// Mitsubishi GX Works2 project: BookEX6_31 Rotation   PLC: Q13UDV

TYPE WordBit : STRUCT
  Data : DWORD;
  Flag : BOOL;
END_STRUCT END_TYPE

// global labels: Global
VAR_GLOBAL
  bVar0 AT M5000 : BOOL;
  abArray0 AT M5010 : ARRAY [0..49] OF BOOL;
  sStr0 AT D5000 : STRING[199];
  sStr1 AT D5100 : STRING[199];
  sStr2 AT D5200 : STRING[199];
  sStr3 AT D5300 : STRING[199];
  sStr4 AT D5400 : STRING[199];
  sStr5 AT D5500 : STRING[199];
  sStr6 AT D5600 : STRING[199];
  sStr7 AT D5700 : STRING[199];
  sStr8 AT D5800 : STRING[199];
  sStr9 AT D5900 : STRING[199];
  iVar0 AT D4500 : INT;
  iVar1 AT D4501 : INT;
  iVar2 AT D4502 : INT;
  iVar3 AT D4503 : INT;
  iVar4 AT D4504 : INT;
  iVar5 AT D4505 : INT;
  iVar6 AT D4506 : INT;
  iVar7 AT D4507 : INT;
  iVar8 AT D4508 : INT;
  iVar9 AT D4509 : INT;
  dVar0 AT D4510 : DINT;
  dVar1 AT D4512 : DINT;
  dVar2 AT D4514 : DINT;
  dVar3 AT D4516 : DINT;
  dVar4 AT D4518 : DINT;
  dVar5 AT D4520 : DINT;
  dVar6 AT D4522 : DINT;
  dVar7 AT D4524 : DINT;
  dVar8 AT D4526 : DINT;
  dVar9 AT D4528 : DINT;
  wVar0 AT D4530 : WORD;
  wVar1 AT D4531 : WORD;
  wVar2 AT D4532 : WORD;
  wVar3 AT D4533 : WORD;
  wVar4 AT D4534 : WORD;
  wVar5 AT D4535 : WORD;
  wVar6 AT D4536 : WORD;
  wVar7 AT D4537 : WORD;
  wVar8 AT D4538 : WORD;
  wVar9 AT D4539 : WORD;
  dwVar0 AT D4540 : DWORD;
  dwVar1 AT D4542 : DWORD;
  dwVar2 AT D4544 : DWORD;
  dwVar3 AT D4546 : DWORD;
  dwVar4 AT D4548 : DWORD;
  dwVar5 AT D4550 : DWORD;
  dwVar6 AT D4552 : DWORD;
  dwVar7 AT D4554 : DWORD;
  dwVar8 AT D4556 : DWORD;
  dwVar9 AT D4558 : DWORD;
  fsVar0 AT D4560 : REAL;
  fsVar1 AT D4562 : REAL;
  fsVar2 AT D4564 : REAL;
  fsVar3 AT D4566 : REAL;
  fsVar4 AT D4568 : REAL;
  fsVar5 AT D4570 : REAL;
  fsVar6 AT D4572 : REAL;
  fsVar7 AT D4574 : REAL;
  fsVar8 AT D4576 : REAL;
  fsVar9 AT D4578 : REAL;
  fdVar0 AT D4580 : LREAL;
  tTime0 AT D4620 : TIME;
  tTime1 AT D4622 : TIME;
  tTime2 AT D4624 : TIME;
  tTime3 AT D4626 : TIME;
  tTime4 AT D4628 : TIME;
  tTime5 AT D4630 : TIME;
  tTime6 AT D4632 : TIME;
  tTime7 AT D4634 : TIME;
  tTime8 AT D4636 : TIME;
  tTime9 AT D4638 : TIME;
  tTime10 AT D4640 : TIME;
  bVar1 AT M5001 : BOOL;
  bVar2 AT M5002 : BOOL;
  bVar3 AT M5003 : BOOL;
  bVar4 AT M5004 : BOOL;
  bVar5 AT M5005 : BOOL;
  bVar6 AT M5006 : BOOL;
  bVar7 AT M5007 : BOOL;
  bVar8 AT M5008 : BOOL;
  bVar9 AT M5009 : BOOL;
  abArray1 AT M5060 : ARRAY [0..49] OF BOOL;
  abArray2 AT M5110 : ARRAY [0..49] OF BOOL;
  abArray3 AT M5160 : ARRAY [0..49] OF BOOL;
  abArray4 AT M5210 : ARRAY [0..49] OF BOOL;
  abArray5 AT M5260 : ARRAY [0..49] OF BOOL;
  abArray6 AT M5310 : ARRAY [0..49] OF BOOL;
  abArray7 AT M5360 : ARRAY [0..49] OF BOOL;
  abArray8 AT M5410 : ARRAY [0..49] OF BOOL;
  abArray9 AT M5460 : ARRAY [0..49] OF BOOL;
  fdVar1 AT D4584 : LREAL;
  fdVar2 AT D4588 : LREAL;
  fdVar3 AT D4592 : LREAL;
  fdVar4 AT D4596 : LREAL;
  fdVar5 AT D4600 : LREAL;
  fdVar6 AT D4604 : LREAL;
  fdVar7 AT D4608 : LREAL;
  fdVar8 AT D4612 : LREAL;
  fdVar9 AT D4616 : LREAL;
  afsPen0 AT D2000 : ARRAY [0..499] OF REAL;
  afsPen1 AT D3000 : ARRAY [0..499] OF REAL;
END_VAR
// user libraries (not included): HMI

FUNCTION BitLoadPos2
VAR_INPUT
  w_IN : WORD;
END_VAR
VAR
  wTmp1 : WORD;
END_VAR
VAR_INPUT
  b_Val : BOOL;
  i_Pos : INT;
  i_No : INT;
END_VAR
VAR
  wTmp2 : WORD;
  wTmp3 : WORD;
END_VAR
;
wTmp1 := HFFFF;
wTmp2 := w_IN;
IF b_Val THEN
	SFR(TRUE, 16 - i_No, wTmp1 );
	ROR(TRUE,  i_Pos, wTmp2);
	wTmp3 := wTmp1 OR wTmp2;
	ROL(TRUE,  i_Pos, wTmp3);
ELSE
	SFL(TRUE,  i_No, wTmp1 );
	ROR(TRUE,  i_Pos, wTmp2);
	wTmp3 := wTmp1 AND wTmp2;
	ROL(TRUE,  i_Pos, wTmp3);
END_IF;
BitLoadPos2 := wTmp3;
END_FUNCTION

FUNCTION dwBitArray
VAR_INPUT
  dwInp : DWORD;
  iOffset : INT;
  iLength : INT;
END_VAR
VAR
  ix : INT;
  dwData : DWORD;
  dwMask : DWORD;
END_VAR
;
dwMask := 0;
FOR ix := 0 TO iLength-1 DO 
	SM700 := TRUE;
	DRCL(TRUE, 1, dwMask); 
END_FOR;
dwData := dwInp;
DROR(TRUE, iOffset, dwData);
dwBitArray := dwData AND dwMask;
END_FUNCTION

PROGRAM ExBitArray
(* structured ladder/FBD written out as ST: instructions are called as NAME(EN, inputs, outputs); _pN, _eN, _tN stand for wires *)
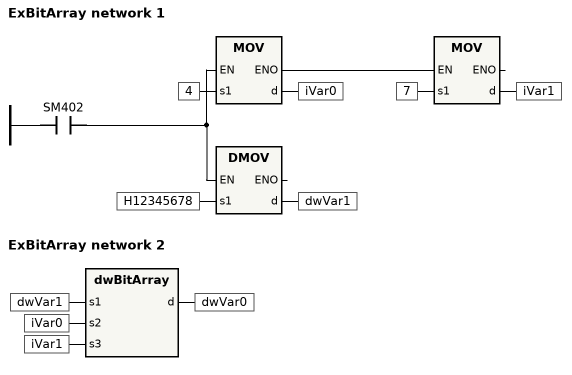
(* network 1 *)
_e1 := MOV(SM402, 4, iVar0);
MOV(_e1, 7, iVar1);
DMOV(SM402, H12345678, dwVar1);
(* network 2 *)
dwVar0 := dwBitArray(dwVar1, iVar0, iVar1);
END_PROGRAM

PROGRAM ExStandard
VAR
  Mov8WORD_1 : Mov8WORD;
  Mov8DWORD_1 : Mov8DWORD;
  wTst0 : WORD;
  wTst1 : WORD;
  wTst2 : WORD;
  wTst3 : WORD;
  wTst4 : WORD;
  dwTst0 : DWORD;
  dwTst1 : DWORD;
  dwTst2 : DWORD;
  dwTst3 : DWORD;
  dwTst4 : DWORD;
  wTst5 : WORD;
  wTst6 : WORD;
  wTst7 : WORD;
  dwTst5 : DWORD;
  dwTst6 : DWORD;
  dwTst7 : DWORD;
END_VAR
(* structured ladder/FBD written out as ST: instructions are called as NAME(EN, inputs, outputs); _pN, _eN, _tN stand for wires *)
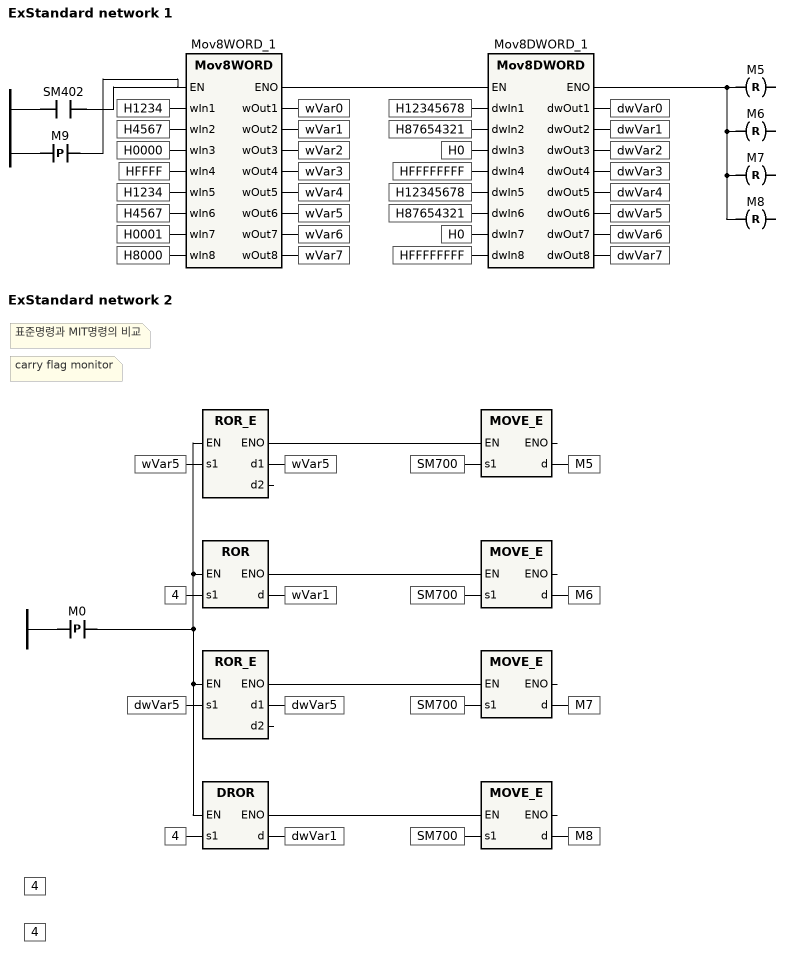
(* network 1 *)
Mov8WORD_1(EN := SM402 OR LDP(TRUE, M9), wIn1 := H1234, wIn2 := H4567, wIn3 := H0000, wIn4 := HFFFF, wIn5 := H1234, wIn6 := H4567, wIn7 := H0001, wIn8 := H8000, wOut1 => wVar0, wOut2 => wVar1, wOut3 => wVar2, wOut4 => wVar3, wOut5 => wVar4, wOut6 => wVar5, wOut7 => wVar6, wOut8 => wVar7);
Mov8DWORD_1(EN := Mov8WORD_1.ENO, dwIn1 := H12345678, dwIn2 := H87654321, dwIn3 := H0, dwIn4 := HFFFFFFFF, dwIn5 := H12345678, dwIn6 := H87654321, dwIn7 := H0, dwIn8 := HFFFFFFFF, dwOut1 => dwVar0, dwOut2 => dwVar1, dwOut3 => dwVar2, dwOut4 => dwVar3, dwOut5 => dwVar4, dwOut6 => dwVar5, dwOut7 => dwVar6, dwOut8 => dwVar7);
RST(Mov8DWORD_1.ENO, M5);
RST(Mov8DWORD_1.ENO, M6);
RST(Mov8DWORD_1.ENO, M7);
RST(Mov8DWORD_1.ENO, M8);
(* network 2 *)
(* 표준명령과 MIT명령의 비교 *)
(* carry flag monitor *)
_p1 := LDP(TRUE, M0);
_e2 := ROR_E(_p1, wVar5, wVar5, _open);
MOVE_E(_e2, SM700, M5);
_e3 := ROR(_p1, 4, wVar1);
MOVE_E(_e3, SM700, M6);
_e4 := ROR_E(_p1, dwVar5, dwVar5, _open);
MOVE_E(_e4, SM700, M7);
_e5 := DROR(_p1, 4, dwVar1);
MOVE_E(_e5, SM700, M8);
(* not connected to any output: 4, 4 *)
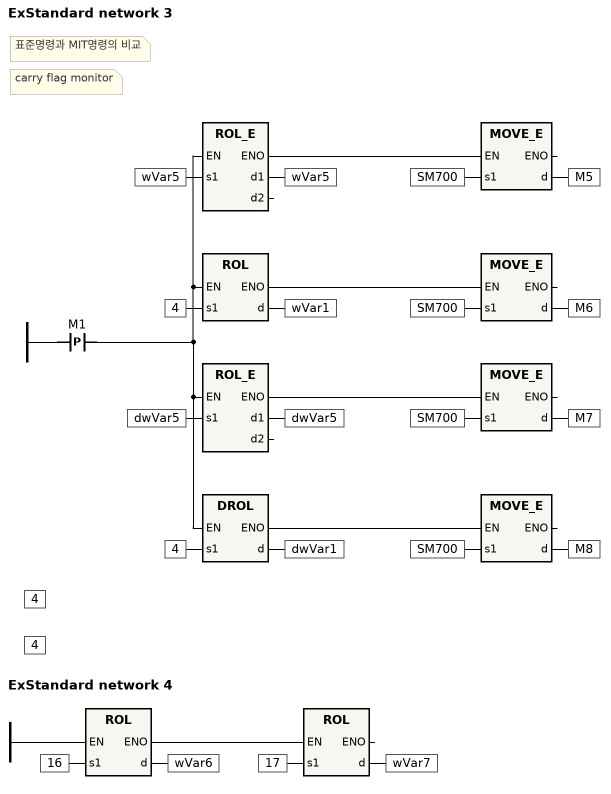
(* network 3 *)
(* 표준명령과 MIT명령의 비교 *)
(* carry flag monitor *)
_p1 := LDP(TRUE, M1);
_e2 := ROL_E(_p1, wVar5, wVar5, _open);
MOVE_E(_e2, SM700, M5);
_e3 := ROL(_p1, 4, wVar1);
MOVE_E(_e3, SM700, M6);
_e4 := ROL_E(_p1, dwVar5, dwVar5, _open);
MOVE_E(_e4, SM700, M7);
_e5 := DROL(_p1, 4, dwVar1);
MOVE_E(_e5, SM700, M8);
(* not connected to any output: 4, 4 *)
(* network 4 *)
_e1 := ROL(TRUE, 16, wVar6);
ROL(_e1, 17, wVar7);
END_PROGRAM

PROGRAM ExDROR
VAR
  Mov8WORD_1 : Mov8WORD;
  Mov8DWORD_1 : Mov8DWORD;
  wTst0 : WORD;
  wTst1 : WORD;
  wTst2 : WORD;
  wTst3 : WORD;
  wTst4 : WORD;
  dwTst0 : DWORD;
  dwTst1 : DWORD;
  dwTst2 : DWORD;
  dwTst3 : DWORD;
  dwTst4 : DWORD;
END_VAR
(* structured ladder/FBD written out as ST: instructions are called as NAME(EN, inputs, outputs); _pN, _eN, _tN stand for wires *)
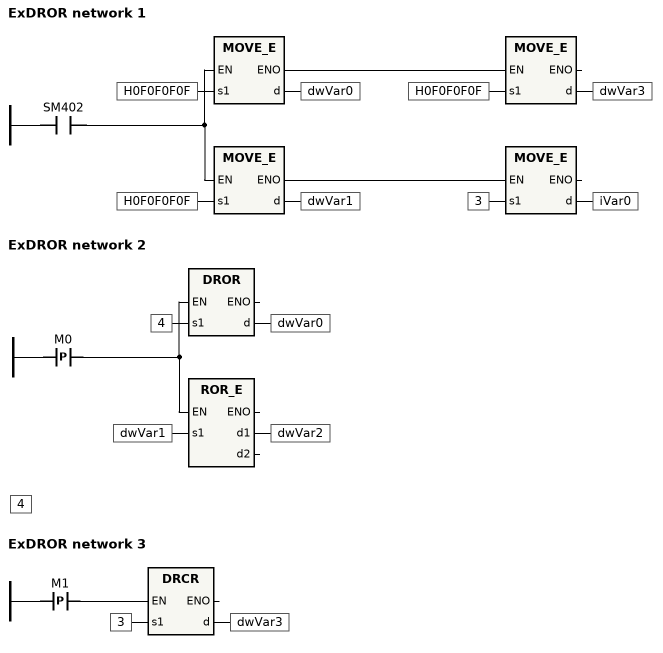
(* network 1 *)
_e1 := MOVE_E(SM402, H0F0F0F0F, dwVar0);
MOVE_E(_e1, H0F0F0F0F, dwVar3);
_e2 := MOVE_E(SM402, H0F0F0F0F, dwVar1);
MOVE_E(_e2, 3, iVar0);
(* network 2 *)
_p1 := LDP(TRUE, M0);
DROR(_p1, 4, dwVar0);
ROR_E(_p1, dwVar1, dwVar2, _open);
(* not connected to any output: 4 *)
(* network 3 *)
DRCR(LDP(TRUE, M1), 3, dwVar3);
END_PROGRAM

PROGRAM ExLib
(* structured ladder/FBD written out as ST: instructions are called as NAME(EN, inputs, outputs); _pN, _eN, _tN stand for wires *)
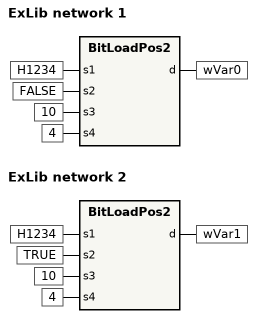
(* network 1 *)
wVar0 := BitLoadPos2(H1234, FALSE, 10, 4);
(* network 2 *)
wVar1 := BitLoadPos2(H1234, TRUE, 10, 4);
END_PROGRAM

PROGRAM ExRingCnt
VAR
  TON_E_1 : TON_E;
  HMI05_1 : HMI05;
END_VAR
(* structured ladder/FBD written out as ST: instructions are called as NAME(EN, inputs, outputs); _pN, _eN, _tN stand for wires *)
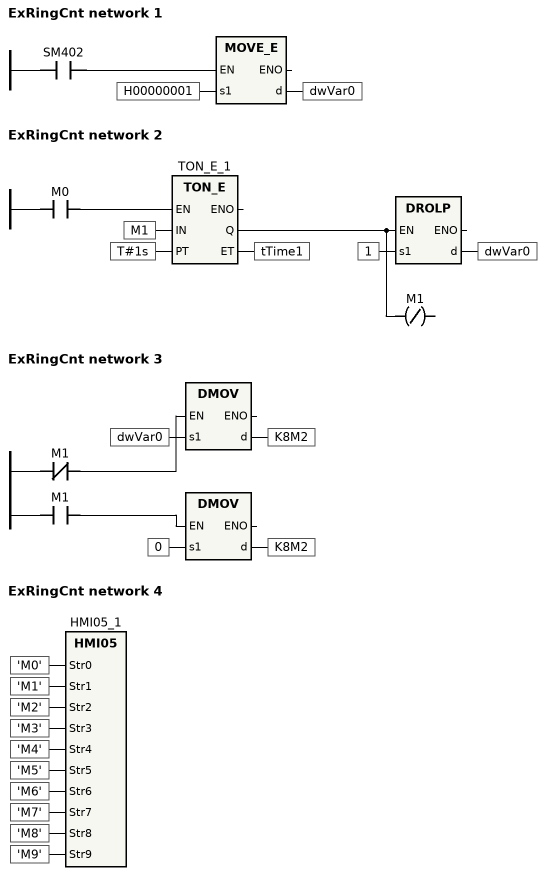
(* network 1 *)
MOVE_E(SM402, H00000001, dwVar0);
(* network 2 *)
TON_E_1(EN := M0, IN := M1, PT := T#1s, ET => tTime1);
M1 := NOT TON_E_1.Q;
DROLP(TON_E_1.Q, 1, dwVar0);
(* network 3 *)
DMOV(NOT M1, dwVar0, K8M2);
DMOV(M1, 0, K8M2);
(* network 4 *)
HMI05_1(Str0 := 'M0', Str1 := 'M1', Str2 := 'M2', Str3 := 'M3', Str4 := 'M4', Str5 := 'M5', Str6 := 'M6', Str7 := 'M7', Str8 := 'M8', Str9 := 'M9');
END_PROGRAM

PROGRAM ExROL
VAR
  Mov8WORD_1 : Mov8WORD;
  Mov8DWORD_1 : Mov8DWORD;
  wTst0 : WORD;
  wTst1 : WORD;
  wTst2 : WORD;
  wTst3 : WORD;
  wTst4 : WORD;
  dwTst0 : DWORD;
  dwTst1 : DWORD;
  dwTst2 : DWORD;
  dwTst3 : DWORD;
  dwTst4 : DWORD;
END_VAR
(* structured ladder/FBD written out as ST: instructions are called as NAME(EN, inputs, outputs); _pN, _eN, _tN stand for wires *)
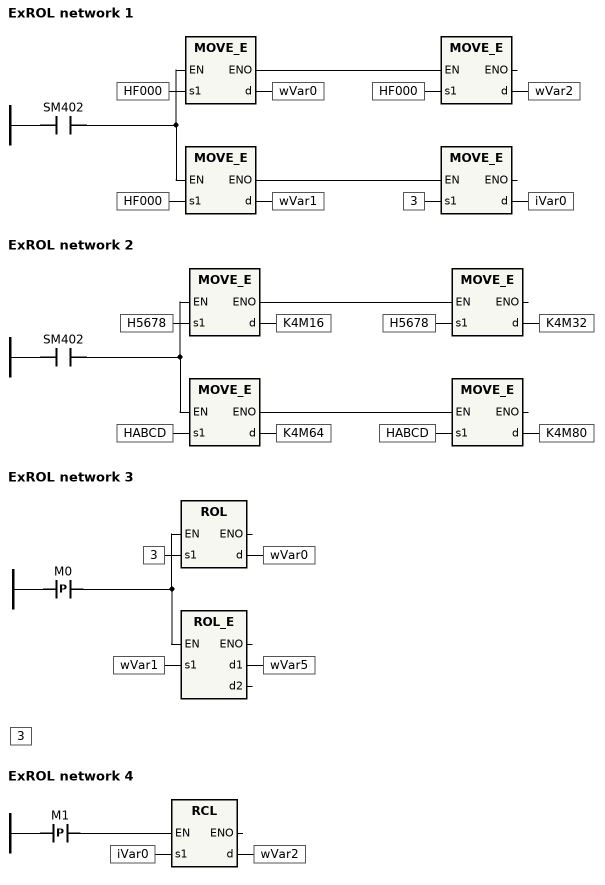
(* network 1 *)
_e1 := MOVE_E(SM402, HF000, wVar0);
MOVE_E(_e1, HF000, wVar2);
_e2 := MOVE_E(SM402, HF000, wVar1);
MOVE_E(_e2, 3, iVar0);
(* network 2 *)
_e1 := MOVE_E(SM402, H5678, K4M16);
MOVE_E(_e1, H5678, K4M32);
_e2 := MOVE_E(SM402, HABCD, K4M64);
MOVE_E(_e2, HABCD, K4M80);
(* network 3 *)
_p1 := LDP(TRUE, M0);
ROL(_p1, 3, wVar0);
ROL_E(_p1, wVar1, wVar5, _open);
(* not connected to any output: 3 *)
(* network 4 *)
RCL(LDP(TRUE, M1), iVar0, wVar2);
END_PROGRAM

PROGRAM ExROR
VAR
  Mov8WORD_1 : Mov8WORD;
  Mov8DWORD_1 : Mov8DWORD;
  wTst0 : WORD;
  wTst1 : WORD;
  wTst2 : WORD;
  wTst3 : WORD;
  wTst4 : WORD;
  dwTst0 : DWORD;
  dwTst1 : DWORD;
  dwTst2 : DWORD;
  dwTst3 : DWORD;
  dwTst4 : DWORD;
END_VAR
(* structured ladder/FBD written out as ST: instructions are called as NAME(EN, inputs, outputs); _pN, _eN, _tN stand for wires *)
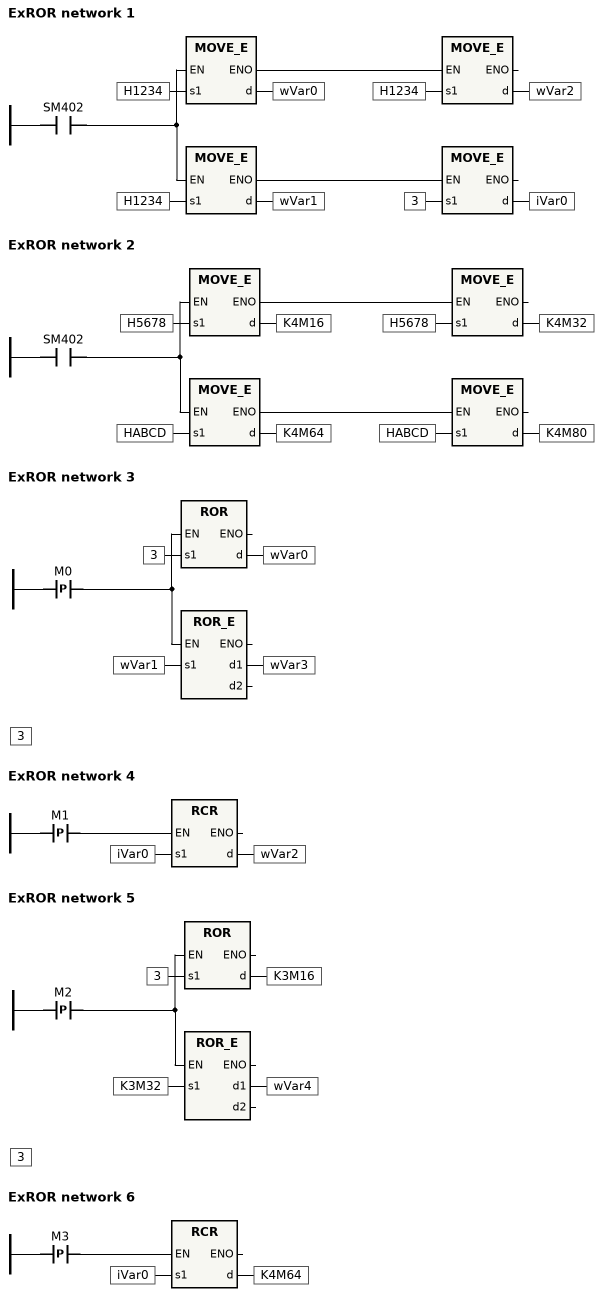
(* network 1 *)
_e1 := MOVE_E(SM402, H1234, wVar0);
MOVE_E(_e1, H1234, wVar2);
_e2 := MOVE_E(SM402, H1234, wVar1);
MOVE_E(_e2, 3, iVar0);
(* network 2 *)
_e1 := MOVE_E(SM402, H5678, K4M16);
MOVE_E(_e1, H5678, K4M32);
_e2 := MOVE_E(SM402, HABCD, K4M64);
MOVE_E(_e2, HABCD, K4M80);
(* network 3 *)
_p1 := LDP(TRUE, M0);
ROR(_p1, 3, wVar0);
ROR_E(_p1, wVar1, wVar3, _open);
(* not connected to any output: 3 *)
(* network 4 *)
RCR(LDP(TRUE, M1), iVar0, wVar2);
(* network 5 *)
_p1 := LDP(TRUE, M2);
ROR(_p1, 3, K3M16);
ROR_E(_p1, K3M32, wVar4, _open);
(* not connected to any output: 3 *)
(* network 6 *)
RCR(LDP(TRUE, M3), iVar0, K4M64);
END_PROGRAM

PROGRAM ExDROL
VAR
  Mov8WORD_1 : Mov8WORD;
  Mov8DWORD_1 : Mov8DWORD;
  wTst0 : WORD;
  wTst1 : WORD;
  wTst2 : WORD;
  wTst3 : WORD;
  wTst4 : WORD;
  dwTst0 : DWORD;
  dwTst1 : DWORD;
  dwTst2 : DWORD;
  dwTst3 : DWORD;
  dwTst4 : DWORD;
  TON_E_1 : TON_E;
END_VAR
(* structured ladder/FBD written out as ST: instructions are called as NAME(EN, inputs, outputs); _pN, _eN, _tN stand for wires *)
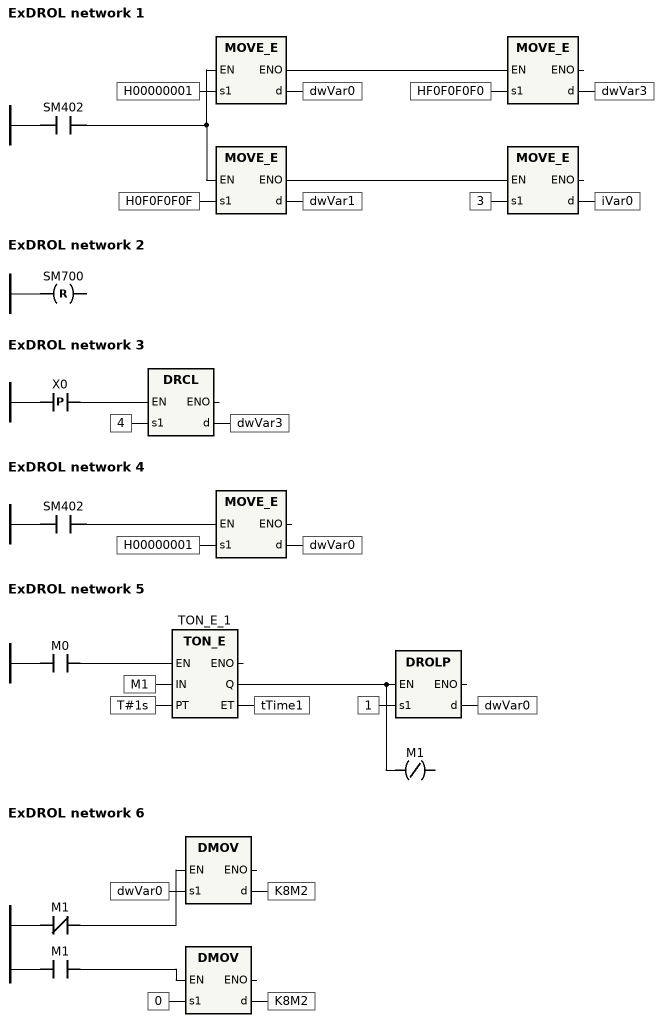
(* network 1 *)
_e1 := MOVE_E(SM402, H00000001, dwVar0);
MOVE_E(_e1, HF0F0F0F0, dwVar3);
_e2 := MOVE_E(SM402, H0F0F0F0F, dwVar1);
MOVE_E(_e2, 3, iVar0);
(* network 2 *)
RST(TRUE, SM700);
(* network 3 *)
DRCL(LDP(TRUE, X0), 4, dwVar3);
(* network 4 *)
MOVE_E(SM402, H00000001, dwVar0);
(* network 5 *)
TON_E_1(EN := M0, IN := M1, PT := T#1s, ET => tTime1);
M1 := NOT TON_E_1.Q;
DROLP(TON_E_1.Q, 1, dwVar0);
(* network 6 *)
DMOV(NOT M1, dwVar0, K8M2);
DMOV(M1, 0, K8M2);
END_PROGRAM
